(* Logix 5000 project; controller RN21_Architecture 1769-L16ER-BB1B rev 35.11; software revision 35.00; part 6 of 9 *)
(* tags used below, declared in another part *)
   AUDSrc : UDT_Audit;
   RN21_AUD_BAMTrig : DINT[5];
   RN21_AUDBAM_ONS : BOOL[128];
   RN21_Map_BAM : BOOL[128];
(* MainProgram, continued *)

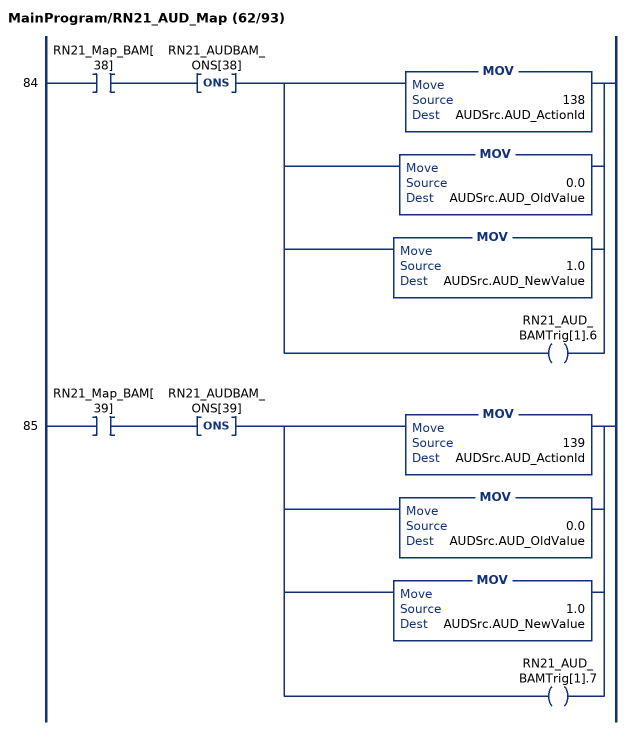
   [picture p144: MainProgram/RN21_AUD_Map rungs 84-85]
   84: XIC(RN21_Map_BAM[38])ONS(RN21_AUDBAM_ONS[38])[MOV(138,AUDSrc.AUD_ActionId) ,MOV(0.0,AUDSrc.AUD_OldValue) ,MOV(1.0,AUDSrc.AUD_NewValue) ,OTE(RN21_AUD_BAMTrig[1].6) ];
   85: XIC(RN21_Map_BAM[39])ONS(RN21_AUDBAM_ONS[39])[MOV(139,AUDSrc.AUD_ActionId) ,MOV(0.0,AUDSrc.AUD_OldValue) ,MOV(1.0,AUDSrc.AUD_NewValue) ,OTE(RN21_AUD_BAMTrig[1].7) ];
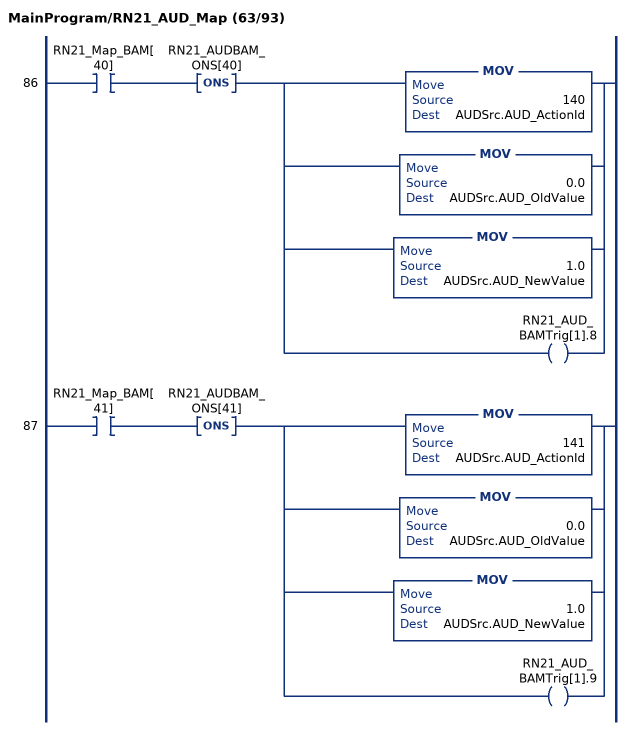
   86: XIC(RN21_Map_BAM[40])ONS(RN21_AUDBAM_ONS[40])[MOV(140,AUDSrc.AUD_ActionId) ,MOV(0.0,AUDSrc.AUD_OldValue) ,MOV(1.0,AUDSrc.AUD_NewValue) ,OTE(RN21_AUD_BAMTrig[1].8) ];
   87: XIC(RN21_Map_BAM[41])ONS(RN21_AUDBAM_ONS[41])[MOV(141,AUDSrc.AUD_ActionId) ,MOV(0.0,AUDSrc.AUD_OldValue) ,MOV(1.0,AUDSrc.AUD_NewValue) ,OTE(RN21_AUD_BAMTrig[1].9) ];
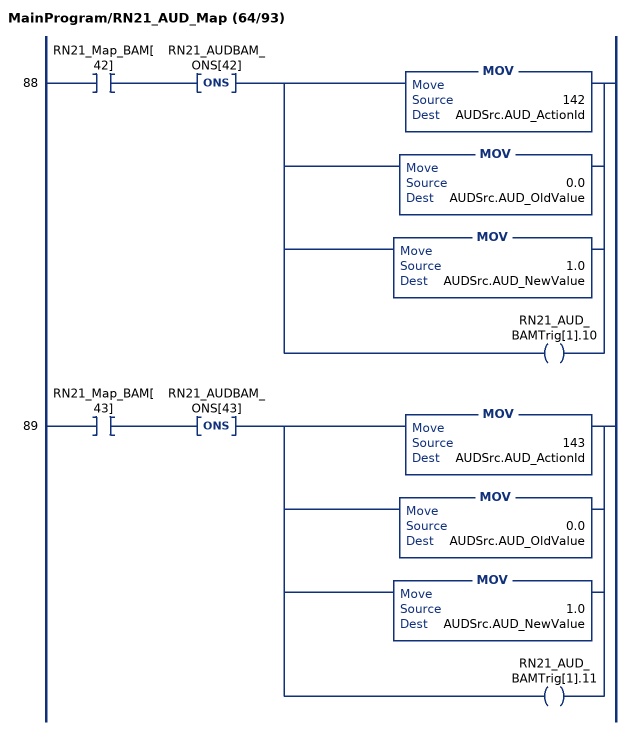
   88: XIC(RN21_Map_BAM[42])ONS(RN21_AUDBAM_ONS[42])[MOV(142,AUDSrc.AUD_ActionId) ,MOV(0.0,AUDSrc.AUD_OldValue) ,MOV(1.0,AUDSrc.AUD_NewValue) ,OTE(RN21_AUD_BAMTrig[1].10) ];
   89: XIC(RN21_Map_BAM[43])ONS(RN21_AUDBAM_ONS[43])[MOV(143,AUDSrc.AUD_ActionId) ,MOV(0.0,AUDSrc.AUD_OldValue) ,MOV(1.0,AUDSrc.AUD_NewValue) ,OTE(RN21_AUD_BAMTrig[1].11) ];
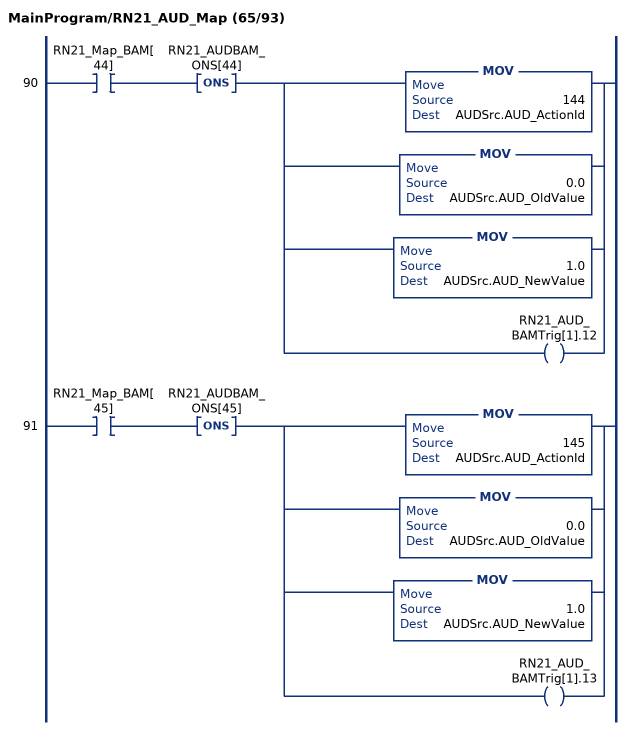
   90: XIC(RN21_Map_BAM[44])ONS(RN21_AUDBAM_ONS[44])[MOV(144,AUDSrc.AUD_ActionId) ,MOV(0.0,AUDSrc.AUD_OldValue) ,MOV(1.0,AUDSrc.AUD_NewValue) ,OTE(RN21_AUD_BAMTrig[1].12) ];
   91: XIC(RN21_Map_BAM[45])ONS(RN21_AUDBAM_ONS[45])[MOV(145,AUDSrc.AUD_ActionId) ,MOV(0.0,AUDSrc.AUD_OldValue) ,MOV(1.0,AUDSrc.AUD_NewValue) ,OTE(RN21_AUD_BAMTrig[1].13) ];
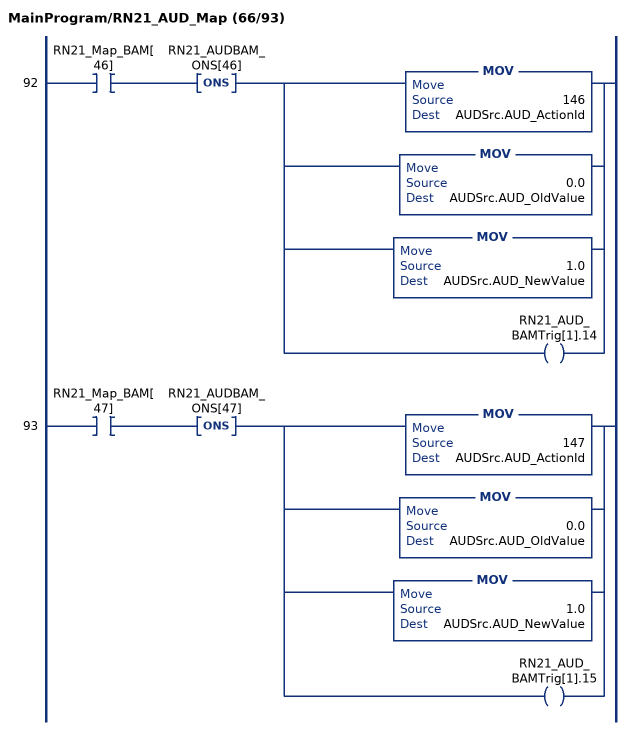
   92: XIC(RN21_Map_BAM[46])ONS(RN21_AUDBAM_ONS[46])[MOV(146,AUDSrc.AUD_ActionId) ,MOV(0.0,AUDSrc.AUD_OldValue) ,MOV(1.0,AUDSrc.AUD_NewValue) ,OTE(RN21_AUD_BAMTrig[1].14) ];
   93: XIC(RN21_Map_BAM[47])ONS(RN21_AUDBAM_ONS[47])[MOV(147,AUDSrc.AUD_ActionId) ,MOV(0.0,AUDSrc.AUD_OldValue) ,MOV(1.0,AUDSrc.AUD_NewValue) ,OTE(RN21_AUD_BAMTrig[1].15) ];
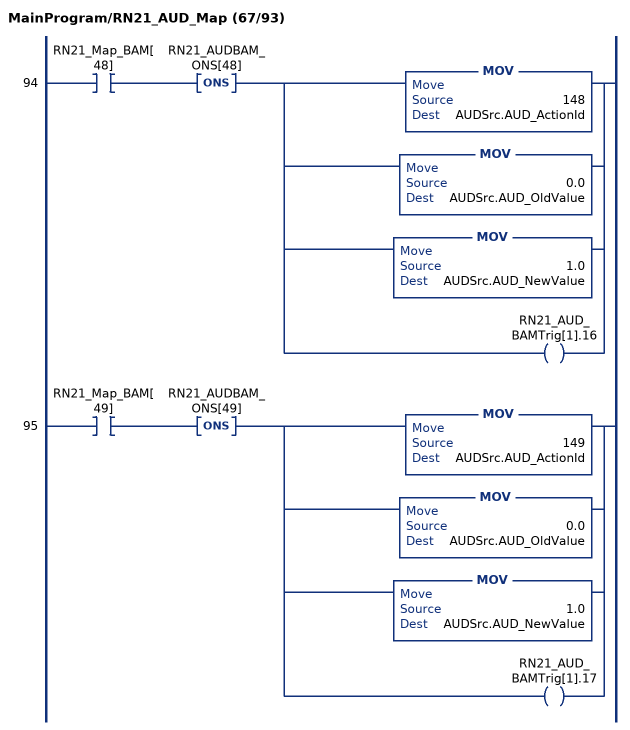
   94: XIC(RN21_Map_BAM[48])ONS(RN21_AUDBAM_ONS[48])[MOV(148,AUDSrc.AUD_ActionId) ,MOV(0.0,AUDSrc.AUD_OldValue) ,MOV(1.0,AUDSrc.AUD_NewValue) ,OTE(RN21_AUD_BAMTrig[1].16) ];
   95: XIC(RN21_Map_BAM[49])ONS(RN21_AUDBAM_ONS[49])[MOV(149,AUDSrc.AUD_ActionId) ,MOV(0.0,AUDSrc.AUD_OldValue) ,MOV(1.0,AUDSrc.AUD_NewValue) ,OTE(RN21_AUD_BAMTrig[1].17) ];
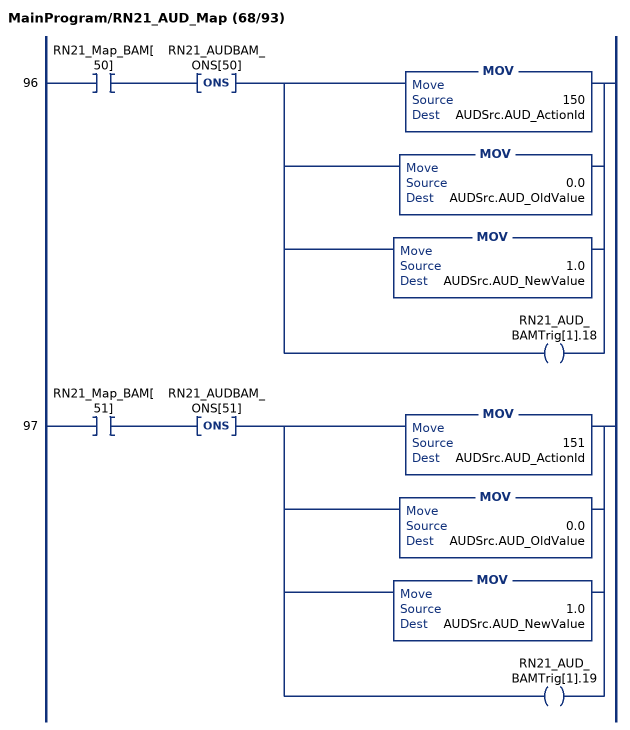
   96: XIC(RN21_Map_BAM[50])ONS(RN21_AUDBAM_ONS[50])[MOV(150,AUDSrc.AUD_ActionId) ,MOV(0.0,AUDSrc.AUD_OldValue) ,MOV(1.0,AUDSrc.AUD_NewValue) ,OTE(RN21_AUD_BAMTrig[1].18) ];
   97: XIC(RN21_Map_BAM[51])ONS(RN21_AUDBAM_ONS[51])[MOV(151,AUDSrc.AUD_ActionId) ,MOV(0.0,AUDSrc.AUD_OldValue) ,MOV(1.0,AUDSrc.AUD_NewValue) ,OTE(RN21_AUD_BAMTrig[1].19) ];
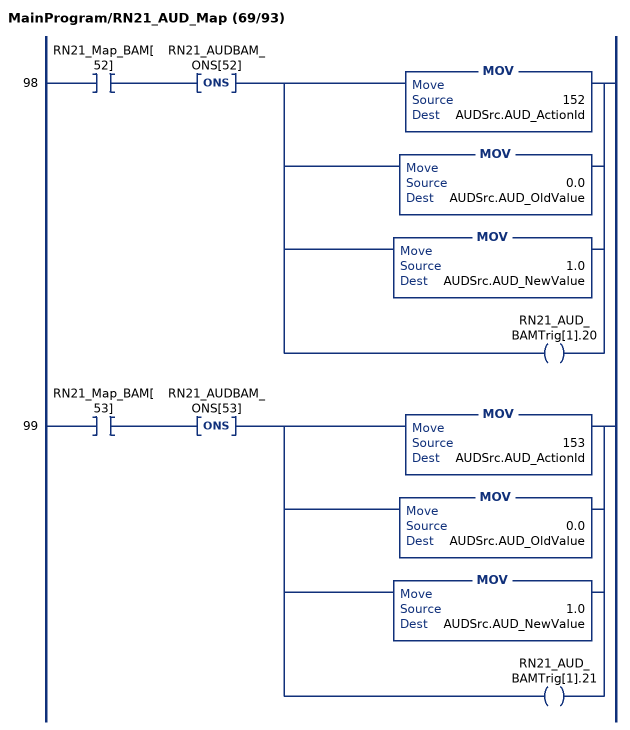
   98: XIC(RN21_Map_BAM[52])ONS(RN21_AUDBAM_ONS[52])[MOV(152,AUDSrc.AUD_ActionId) ,MOV(0.0,AUDSrc.AUD_OldValue) ,MOV(1.0,AUDSrc.AUD_NewValue) ,OTE(RN21_AUD_BAMTrig[1].20) ];
   99: XIC(RN21_Map_BAM[53])ONS(RN21_AUDBAM_ONS[53])[MOV(153,AUDSrc.AUD_ActionId) ,MOV(0.0,AUDSrc.AUD_OldValue) ,MOV(1.0,AUDSrc.AUD_NewValue) ,OTE(RN21_AUD_BAMTrig[1].21) ];
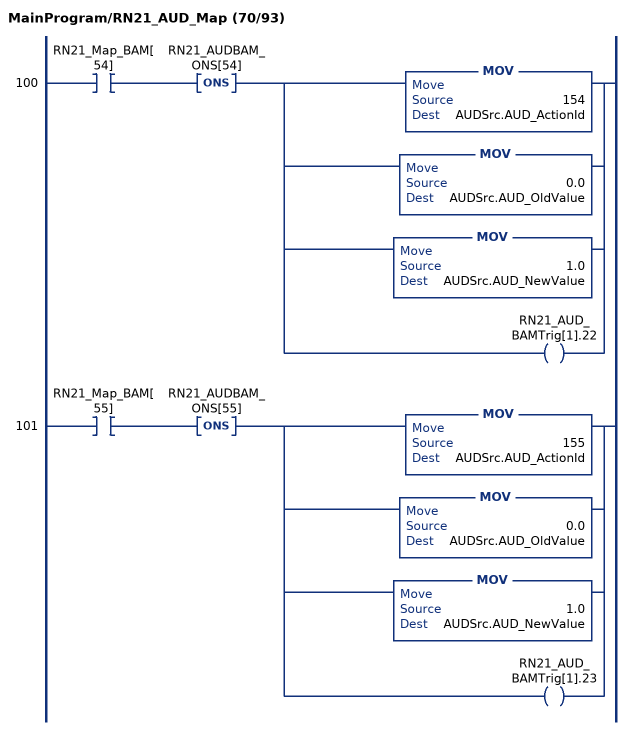
   100: XIC(RN21_Map_BAM[54])ONS(RN21_AUDBAM_ONS[54])[MOV(154,AUDSrc.AUD_ActionId) ,MOV(0.0,AUDSrc.AUD_OldValue) ,MOV(1.0,AUDSrc.AUD_NewValue) ,OTE(RN21_AUD_BAMTrig[1].22) ];
   101: XIC(RN21_Map_BAM[55])ONS(RN21_AUDBAM_ONS[55])[MOV(155,AUDSrc.AUD_ActionId) ,MOV(0.0,AUDSrc.AUD_OldValue) ,MOV(1.0,AUDSrc.AUD_NewValue) ,OTE(RN21_AUD_BAMTrig[1].23) ];
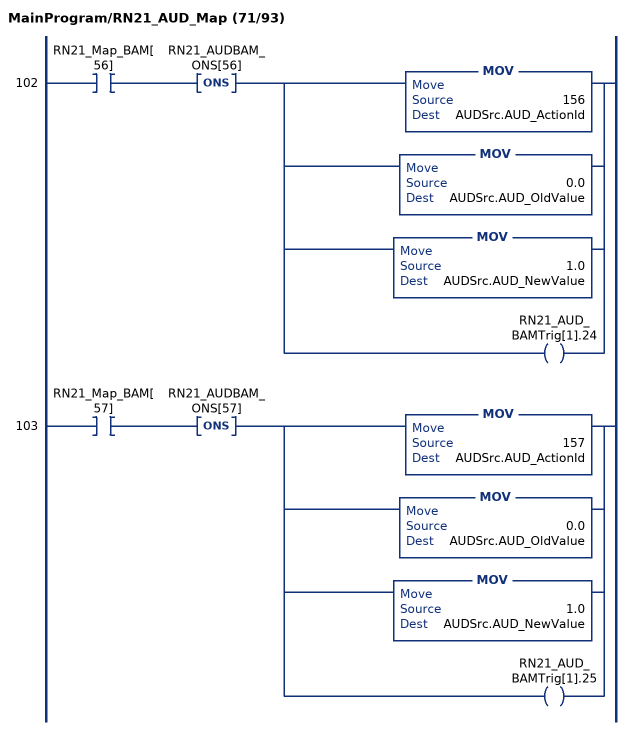
   102: XIC(RN21_Map_BAM[56])ONS(RN21_AUDBAM_ONS[56])[MOV(156,AUDSrc.AUD_ActionId) ,MOV(0.0,AUDSrc.AUD_OldValue) ,MOV(1.0,AUDSrc.AUD_NewValue) ,OTE(RN21_AUD_BAMTrig[1].24) ];
   103: XIC(RN21_Map_BAM[57])ONS(RN21_AUDBAM_ONS[57])[MOV(157,AUDSrc.AUD_ActionId) ,MOV(0.0,AUDSrc.AUD_OldValue) ,MOV(1.0,AUDSrc.AUD_NewValue) ,OTE(RN21_AUD_BAMTrig[1].25) ];
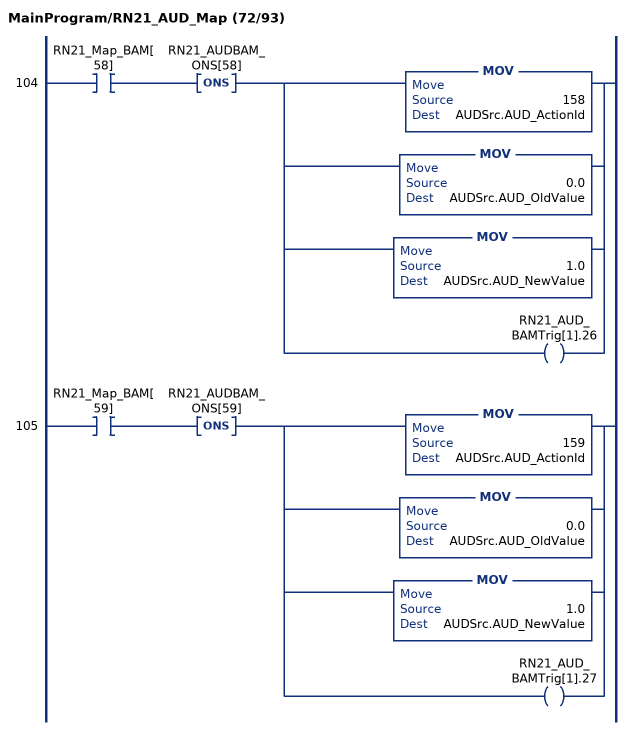
   104: XIC(RN21_Map_BAM[58])ONS(RN21_AUDBAM_ONS[58])[MOV(158,AUDSrc.AUD_ActionId) ,MOV(0.0,AUDSrc.AUD_OldValue) ,MOV(1.0,AUDSrc.AUD_NewValue) ,OTE(RN21_AUD_BAMTrig[1].26) ];
   105: XIC(RN21_Map_BAM[59])ONS(RN21_AUDBAM_ONS[59])[MOV(159,AUDSrc.AUD_ActionId) ,MOV(0.0,AUDSrc.AUD_OldValue) ,MOV(1.0,AUDSrc.AUD_NewValue) ,OTE(RN21_AUD_BAMTrig[1].27) ];
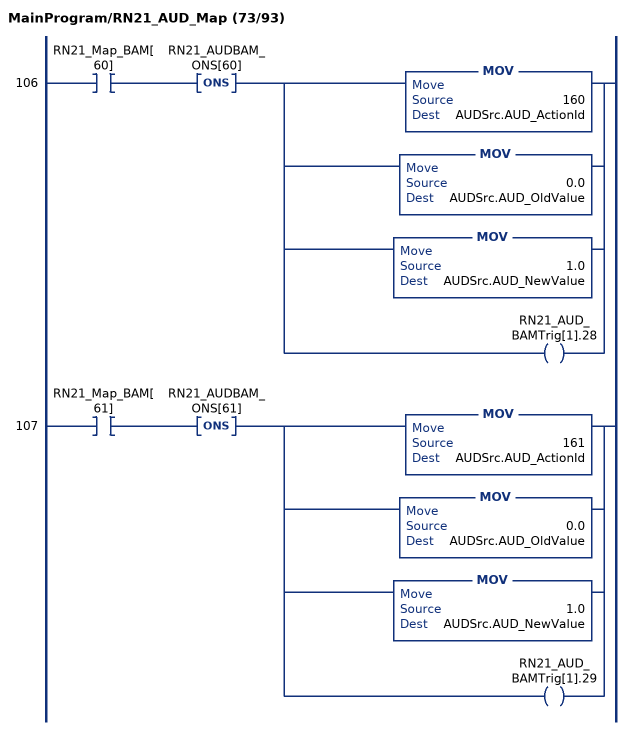
   106: XIC(RN21_Map_BAM[60])ONS(RN21_AUDBAM_ONS[60])[MOV(160,AUDSrc.AUD_ActionId) ,MOV(0.0,AUDSrc.AUD_OldValue) ,MOV(1.0,AUDSrc.AUD_NewValue) ,OTE(RN21_AUD_BAMTrig[1].28) ];
   107: XIC(RN21_Map_BAM[61])ONS(RN21_AUDBAM_ONS[61])[MOV(161,AUDSrc.AUD_ActionId) ,MOV(0.0,AUDSrc.AUD_OldValue) ,MOV(1.0,AUDSrc.AUD_NewValue) ,OTE(RN21_AUD_BAMTrig[1].29) ];
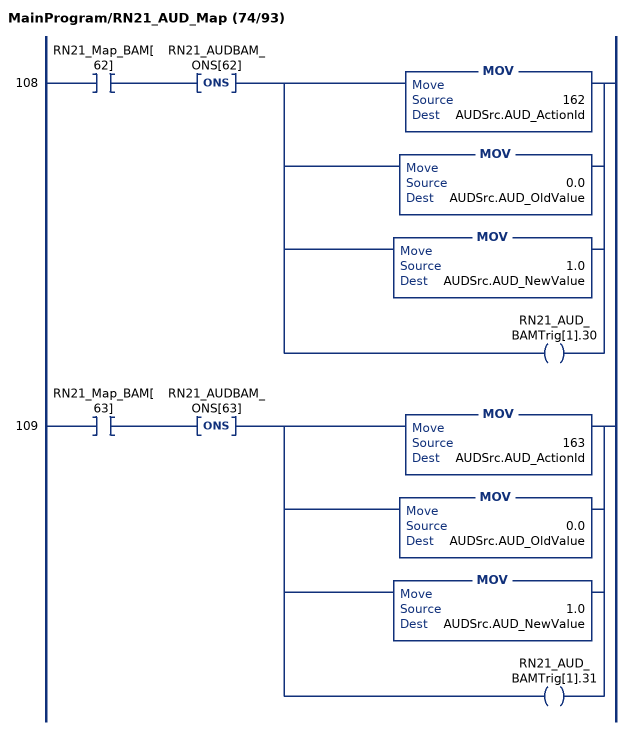
   108: XIC(RN21_Map_BAM[62])ONS(RN21_AUDBAM_ONS[62])[MOV(162,AUDSrc.AUD_ActionId) ,MOV(0.0,AUDSrc.AUD_OldValue) ,MOV(1.0,AUDSrc.AUD_NewValue) ,OTE(RN21_AUD_BAMTrig[1].30) ];
   109: XIC(RN21_Map_BAM[63])ONS(RN21_AUDBAM_ONS[63])[MOV(163,AUDSrc.AUD_ActionId) ,MOV(0.0,AUDSrc.AUD_OldValue) ,MOV(1.0,AUDSrc.AUD_NewValue) ,OTE(RN21_AUD_BAMTrig[1].31) ];
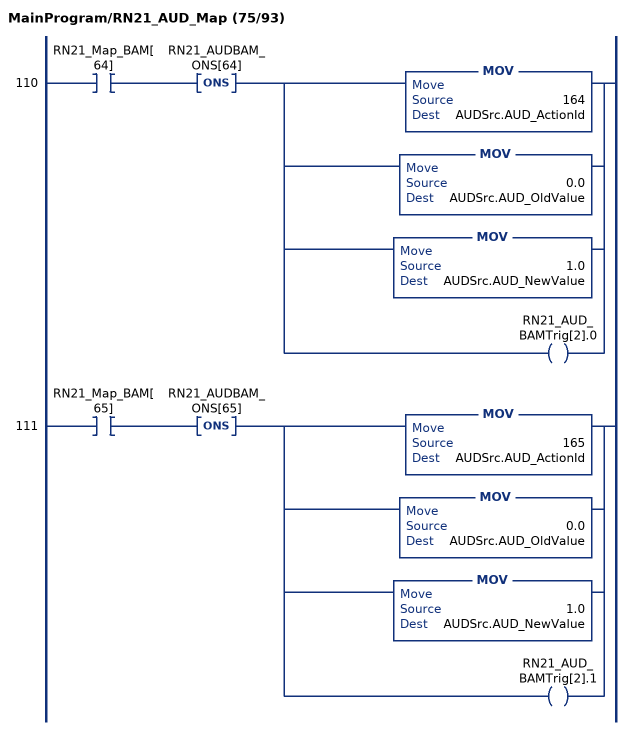
   110: XIC(RN21_Map_BAM[64])ONS(RN21_AUDBAM_ONS[64])[MOV(164,AUDSrc.AUD_ActionId) ,MOV(0.0,AUDSrc.AUD_OldValue) ,MOV(1.0,AUDSrc.AUD_NewValue) ,OTE(RN21_AUD_BAMTrig[2].0) ];
   111: XIC(RN21_Map_BAM[65])ONS(RN21_AUDBAM_ONS[65])[MOV(165,AUDSrc.AUD_ActionId) ,MOV(0.0,AUDSrc.AUD_OldValue) ,MOV(1.0,AUDSrc.AUD_NewValue) ,OTE(RN21_AUD_BAMTrig[2].1) ];
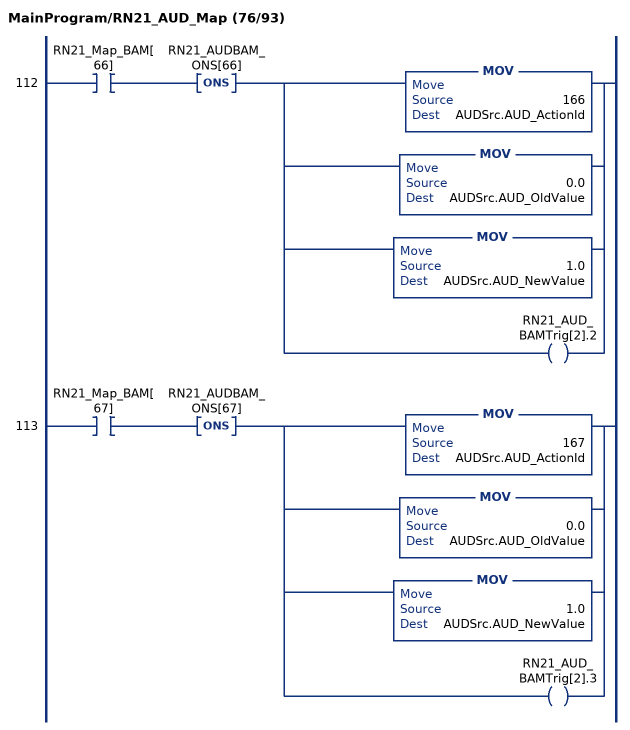
   112: XIC(RN21_Map_BAM[66])ONS(RN21_AUDBAM_ONS[66])[MOV(166,AUDSrc.AUD_ActionId) ,MOV(0.0,AUDSrc.AUD_OldValue) ,MOV(1.0,AUDSrc.AUD_NewValue) ,OTE(RN21_AUD_BAMTrig[2].2) ];
   113: XIC(RN21_Map_BAM[67])ONS(RN21_AUDBAM_ONS[67])[MOV(167,AUDSrc.AUD_ActionId) ,MOV(0.0,AUDSrc.AUD_OldValue) ,MOV(1.0,AUDSrc.AUD_NewValue) ,OTE(RN21_AUD_BAMTrig[2].3) ];
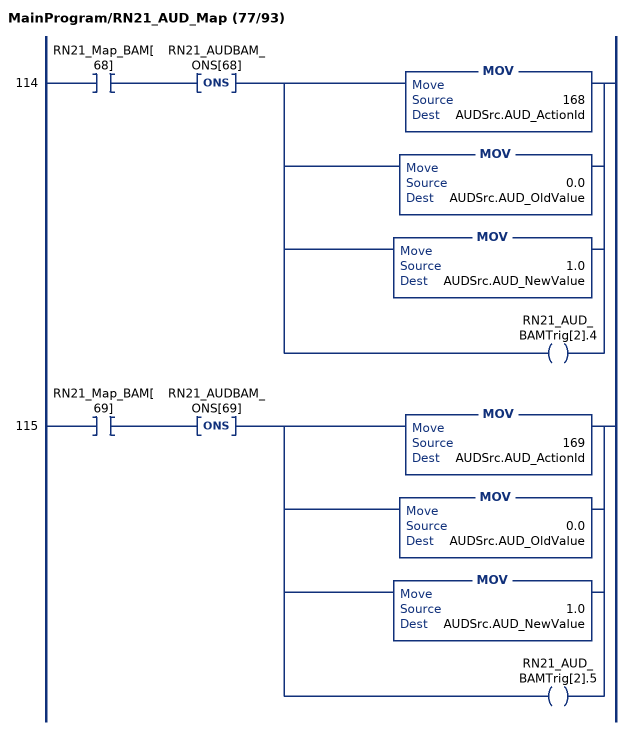
   114: XIC(RN21_Map_BAM[68])ONS(RN21_AUDBAM_ONS[68])[MOV(168,AUDSrc.AUD_ActionId) ,MOV(0.0,AUDSrc.AUD_OldValue) ,MOV(1.0,AUDSrc.AUD_NewValue) ,OTE(RN21_AUD_BAMTrig[2].4) ];
   115: XIC(RN21_Map_BAM[69])ONS(RN21_AUDBAM_ONS[69])[MOV(169,AUDSrc.AUD_ActionId) ,MOV(0.0,AUDSrc.AUD_OldValue) ,MOV(1.0,AUDSrc.AUD_NewValue) ,OTE(RN21_AUD_BAMTrig[2].5) ];
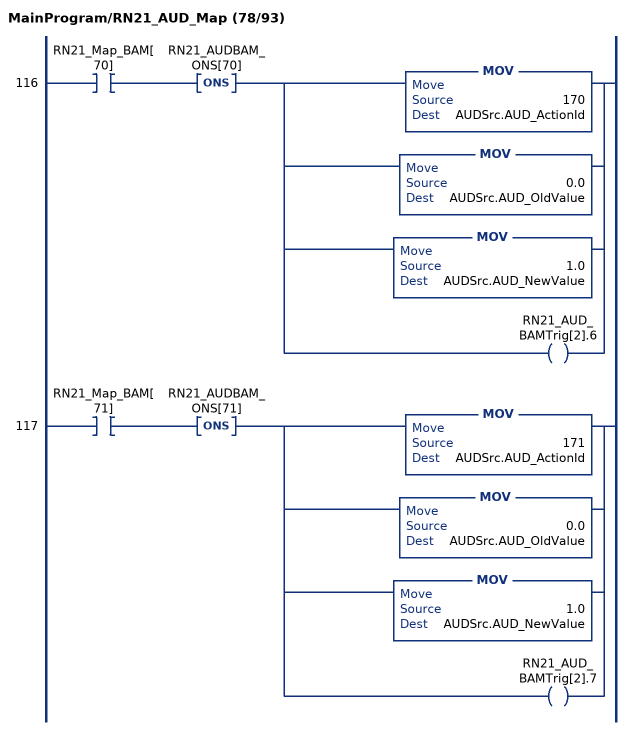
   116: XIC(RN21_Map_BAM[70])ONS(RN21_AUDBAM_ONS[70])[MOV(170,AUDSrc.AUD_ActionId) ,MOV(0.0,AUDSrc.AUD_OldValue) ,MOV(1.0,AUDSrc.AUD_NewValue) ,OTE(RN21_AUD_BAMTrig[2].6) ];
   117: XIC(RN21_Map_BAM[71])ONS(RN21_AUDBAM_ONS[71])[MOV(171,AUDSrc.AUD_ActionId) ,MOV(0.0,AUDSrc.AUD_OldValue) ,MOV(1.0,AUDSrc.AUD_NewValue) ,OTE(RN21_AUD_BAMTrig[2].7) ];
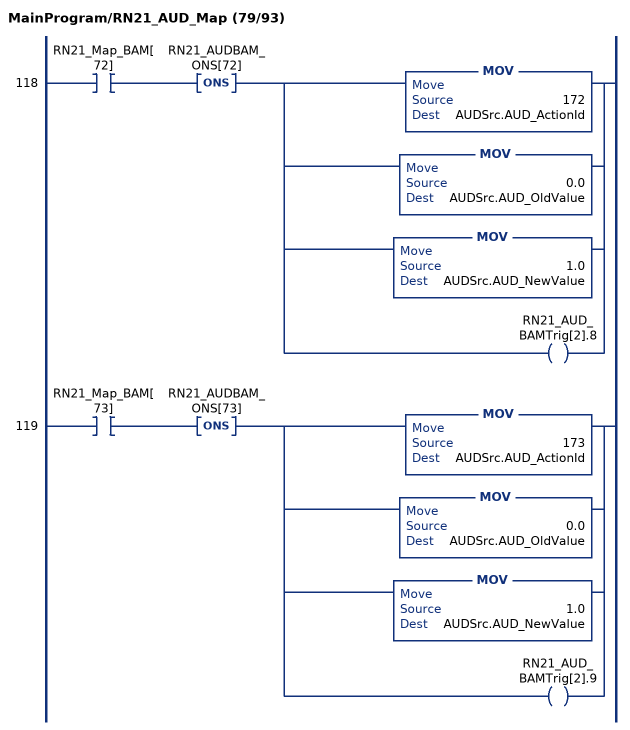
   118: XIC(RN21_Map_BAM[72])ONS(RN21_AUDBAM_ONS[72])[MOV(172,AUDSrc.AUD_ActionId) ,MOV(0.0,AUDSrc.AUD_OldValue) ,MOV(1.0,AUDSrc.AUD_NewValue) ,OTE(RN21_AUD_BAMTrig[2].8) ];
   119: XIC(RN21_Map_BAM[73])ONS(RN21_AUDBAM_ONS[73])[MOV(173,AUDSrc.AUD_ActionId) ,MOV(0.0,AUDSrc.AUD_OldValue) ,MOV(1.0,AUDSrc.AUD_NewValue) ,OTE(RN21_AUD_BAMTrig[2].9) ];
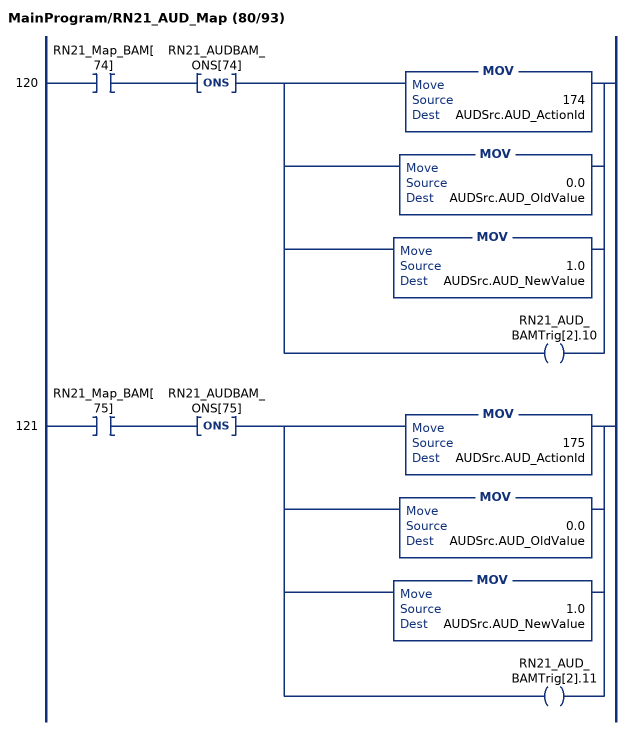
   120: XIC(RN21_Map_BAM[74])ONS(RN21_AUDBAM_ONS[74])[MOV(174,AUDSrc.AUD_ActionId) ,MOV(0.0,AUDSrc.AUD_OldValue) ,MOV(1.0,AUDSrc.AUD_NewValue) ,OTE(RN21_AUD_BAMTrig[2].10) ];
   121: XIC(RN21_Map_BAM[75])ONS(RN21_AUDBAM_ONS[75])[MOV(175,AUDSrc.AUD_ActionId) ,MOV(0.0,AUDSrc.AUD_OldValue) ,MOV(1.0,AUDSrc.AUD_NewValue) ,OTE(RN21_AUD_BAMTrig[2].11) ];
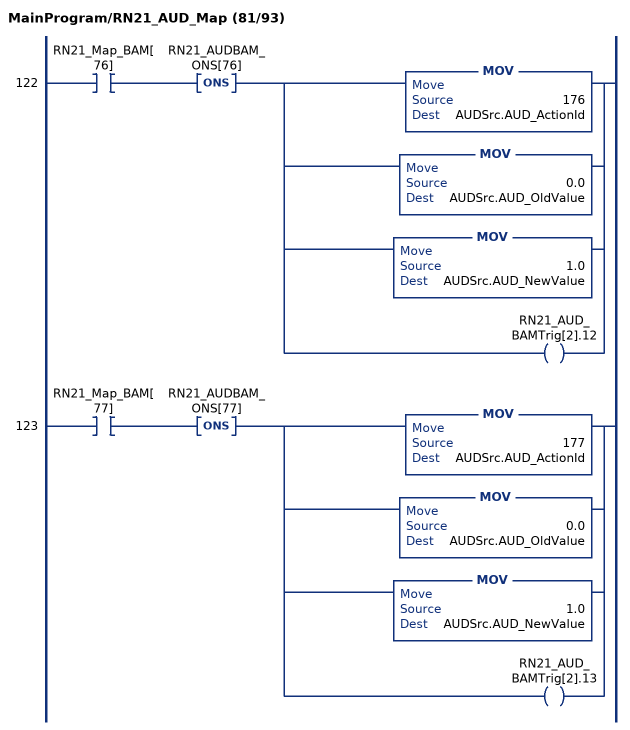
   122: XIC(RN21_Map_BAM[76])ONS(RN21_AUDBAM_ONS[76])[MOV(176,AUDSrc.AUD_ActionId) ,MOV(0.0,AUDSrc.AUD_OldValue) ,MOV(1.0,AUDSrc.AUD_NewValue) ,OTE(RN21_AUD_BAMTrig[2].12) ];
   123: XIC(RN21_Map_BAM[77])ONS(RN21_AUDBAM_ONS[77])[MOV(177,AUDSrc.AUD_ActionId) ,MOV(0.0,AUDSrc.AUD_OldValue) ,MOV(1.0,AUDSrc.AUD_NewValue) ,OTE(RN21_AUD_BAMTrig[2].13) ];
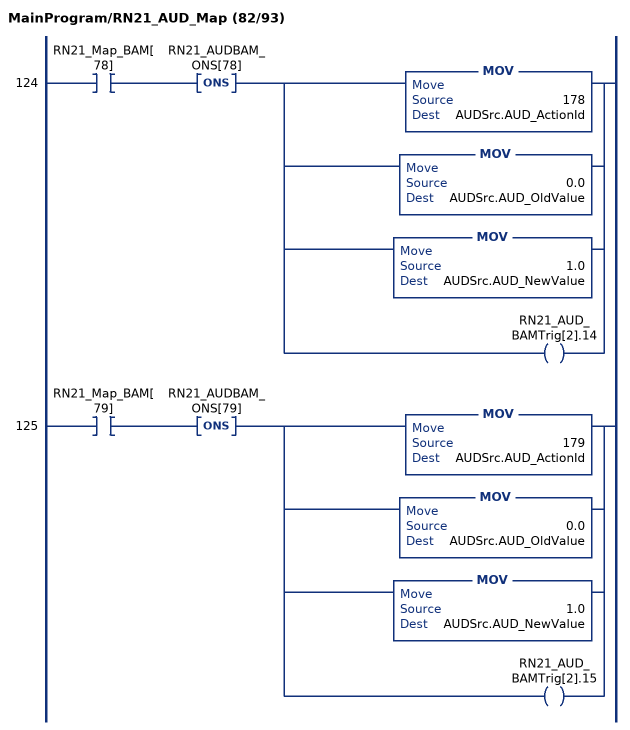
   124: XIC(RN21_Map_BAM[78])ONS(RN21_AUDBAM_ONS[78])[MOV(178,AUDSrc.AUD_ActionId) ,MOV(0.0,AUDSrc.AUD_OldValue) ,MOV(1.0,AUDSrc.AUD_NewValue) ,OTE(RN21_AUD_BAMTrig[2].14) ];
   125: XIC(RN21_Map_BAM[79])ONS(RN21_AUDBAM_ONS[79])[MOV(179,AUDSrc.AUD_ActionId) ,MOV(0.0,AUDSrc.AUD_OldValue) ,MOV(1.0,AUDSrc.AUD_NewValue) ,OTE(RN21_AUD_BAMTrig[2].15) ];
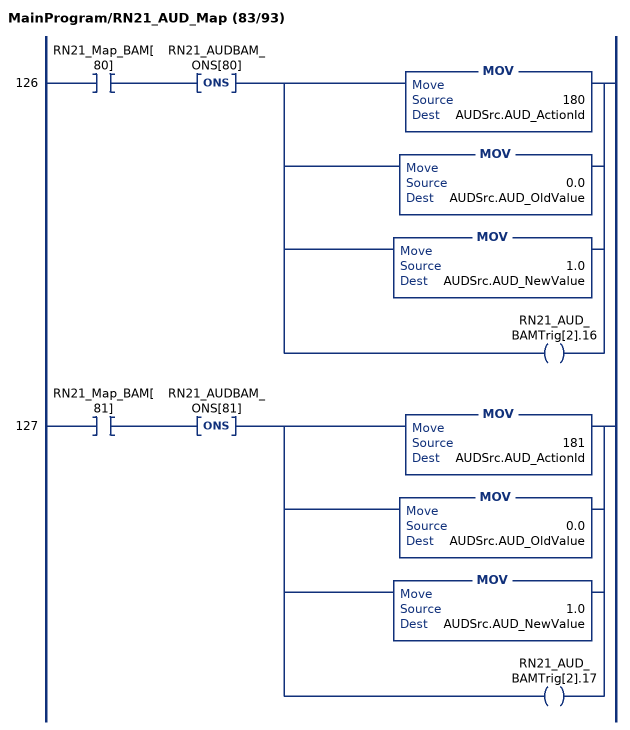
   126: XIC(RN21_Map_BAM[80])ONS(RN21_AUDBAM_ONS[80])[MOV(180,AUDSrc.AUD_ActionId) ,MOV(0.0,AUDSrc.AUD_OldValue) ,MOV(1.0,AUDSrc.AUD_NewValue) ,OTE(RN21_AUD_BAMTrig[2].16) ];
   127: XIC(RN21_Map_BAM[81])ONS(RN21_AUDBAM_ONS[81])[MOV(181,AUDSrc.AUD_ActionId) ,MOV(0.0,AUDSrc.AUD_OldValue) ,MOV(1.0,AUDSrc.AUD_NewValue) ,OTE(RN21_AUD_BAMTrig[2].17) ];
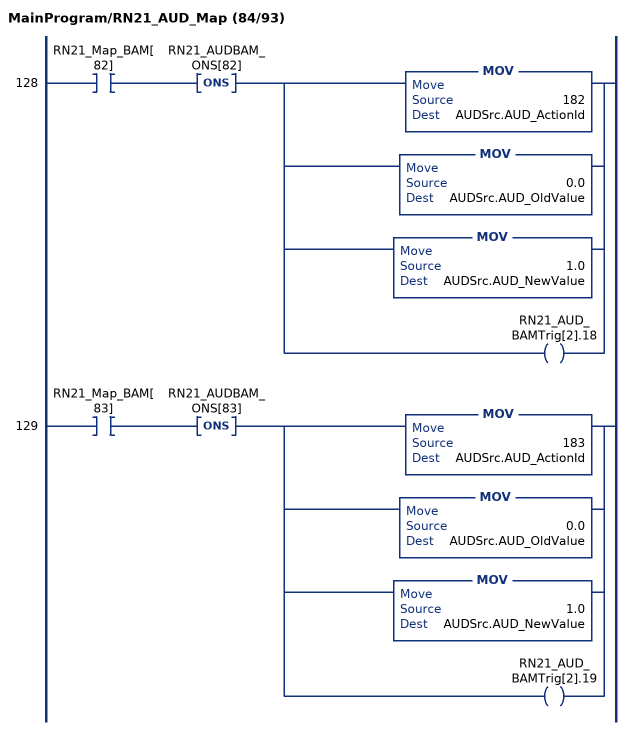
   128: XIC(RN21_Map_BAM[82])ONS(RN21_AUDBAM_ONS[82])[MOV(182,AUDSrc.AUD_ActionId) ,MOV(0.0,AUDSrc.AUD_OldValue) ,MOV(1.0,AUDSrc.AUD_NewValue) ,OTE(RN21_AUD_BAMTrig[2].18) ];
   129: XIC(RN21_Map_BAM[83])ONS(RN21_AUDBAM_ONS[83])[MOV(183,AUDSrc.AUD_ActionId) ,MOV(0.0,AUDSrc.AUD_OldValue) ,MOV(1.0,AUDSrc.AUD_NewValue) ,OTE(RN21_AUD_BAMTrig[2].19) ];
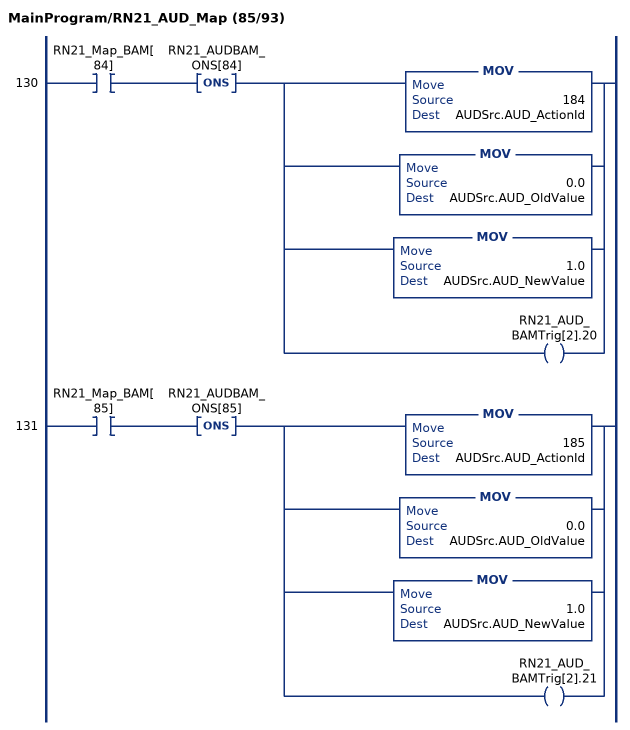
   130: XIC(RN21_Map_BAM[84])ONS(RN21_AUDBAM_ONS[84])[MOV(184,AUDSrc.AUD_ActionId) ,MOV(0.0,AUDSrc.AUD_OldValue) ,MOV(1.0,AUDSrc.AUD_NewValue) ,OTE(RN21_AUD_BAMTrig[2].20) ];
   131: XIC(RN21_Map_BAM[85])ONS(RN21_AUDBAM_ONS[85])[MOV(185,AUDSrc.AUD_ActionId) ,MOV(0.0,AUDSrc.AUD_OldValue) ,MOV(1.0,AUDSrc.AUD_NewValue) ,OTE(RN21_AUD_BAMTrig[2].21) ];
